// TIA Portal V20 export
// export: Created 2026-04-11T06:02:30.5517872Z, ExportSetting WithDefaults, DisplayName Totally Integrated Automation Portal, DisplayVersion V20, DisplayName TIA Portal Openness, DisplayVersion V20, DisplayName TIA Portal Version Control Interface, DisplayVersion V20, DisplayName STEP 7 Professional, DisplayVersion V20, DisplayName STEP 7 Safety, DisplayVersion V20, DisplayName WinCC Basic/Comfort/Advanced, DisplayVersion V20, DisplayName WinCC Unified, DisplayVersion V20
TYPE "udtHMI_SystemRunControl"
// stored: IsFailsafeCompliant false
   STRUCT
      bRunning { ExternalWritable := 'False'} : Bool;
      bPB_Start : Bool;
      bPBEN_Start { ExternalWritable := 'False'} : Bool;
      bPB_Stop : Bool;
      bPBEN_Stop { ExternalWritable := 'False'} : Bool;
   END_STRUCT;
END_TYPE
